# EPICS autosave request: iocBoot/iocBPMRFFE/auto_settings.req
file "BPMRFFE_settings.req",          P=$(P)
